// Mitsubishi GX Works2 project: Project   PLC: Q03UDV

PROGRAM MAIN
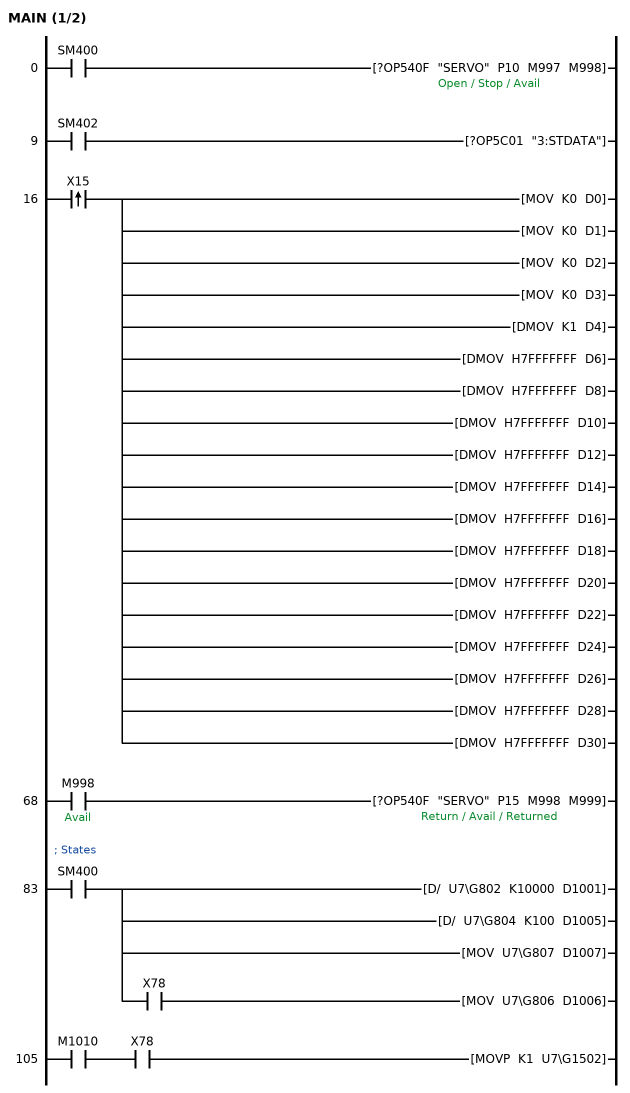
0     LD      SM400
      ?OP540F "SERVO" P10 M997 M998  ; Open / Stop / Avail
9     LD      SM402
      ?OP5C01 "3:STDATA"
16    LDP     X15
      MOV     K0 D0
      MOV     K0 D1
      MOV     K0 D2
      MOV     K0 D3
      DMOV    K1 D4
      DMOV    H7FFFFFFF D6
      DMOV    H7FFFFFFF D8
      DMOV    H7FFFFFFF D10
      DMOV    H7FFFFFFF D12
      DMOV    H7FFFFFFF D14
      DMOV    H7FFFFFFF D16
      DMOV    H7FFFFFFF D18
      DMOV    H7FFFFFFF D20
      DMOV    H7FFFFFFF D22
      DMOV    H7FFFFFFF D24
      DMOV    H7FFFFFFF D26
      DMOV    H7FFFFFFF D28
      DMOV    H7FFFFFFF D30
68    LD      M998  ; Avail
      ?OP540F "SERVO" P15 M998 M999  ; Return / Returned
; States
83    LD      SM400
      D/      U7\G802 K10000 D1001
      D/      U7\G804 K100 D1005
      MOV     U7\G807 D1007
      AND     X78
      MOV     U7\G806 D1006
105   LD      M1010
      AND     X78
      MOVP    K1 U7\G1502
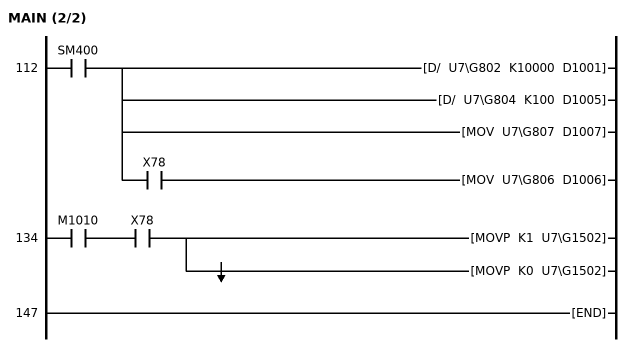
112   LD      SM400
      D/      U7\G802 K10000 D1001
      D/      U7\G804 K100 D1005
      MOV     U7\G807 D1007
      AND     X78
      MOV     U7\G806 D1006
134   LD      M1010
      AND     X78
      MOVP    K1 U7\G1502
      MEF
      MOVP    K0 U7\G1502
147   END
END_PROGRAM

PROGRAM SERVO
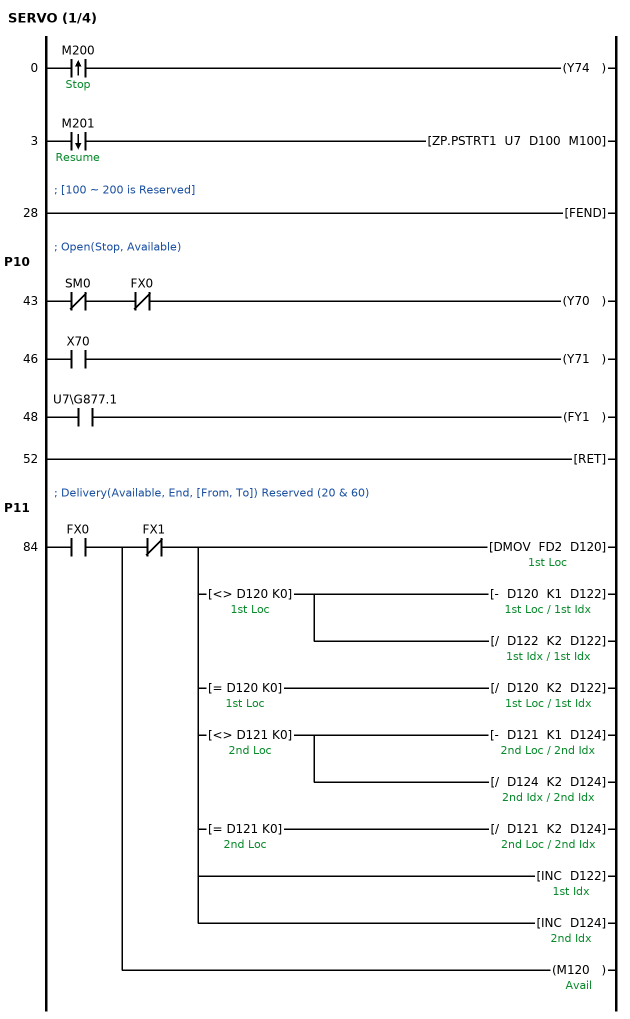
0     LDP     M200  ; Stop
      OUT     Y74
3     LDF     M201  ; Resume
      ZP.PSTRT1 U7 D100 M100
; [100 ~ 200 is Reserved]
28    FEND
      P10
; Open(Stop, Available)
43    LDI     SM0
      ANI     FX0
      OUT     Y70
46    LD      X70
      OUT     Y71
48    LD      U7\G877.1
      OUT     FY1
52    RET
      P11
; Delivery(Available, End, [From, To]) Reserved (20 & 60)
84    LD      FX0
      MPS
      ANI     FX1
      DMOV    FD2 D120  ; 1st Loc
      MPS
      AND<>   D120 K0  ; 1st Loc
      -       D120 K1 D122  ; 1st Idx
      /       D122 K2 D122
      MRD
      AND=    D120 K0  ; 1st Loc
      /       D120 K2 D122
      MRD
      AND<>   D121 K0  ; 2nd Loc
      -       D121 K1 D124  ; 2nd Idx
      /       D124 K2 D124
      MRD
      AND=    D121 K0  ; 2nd Loc
      /       D121 K2 D124
      MPP
      INC     D122
      INC     D124
      MPP
      OUT     M120  ; Avail
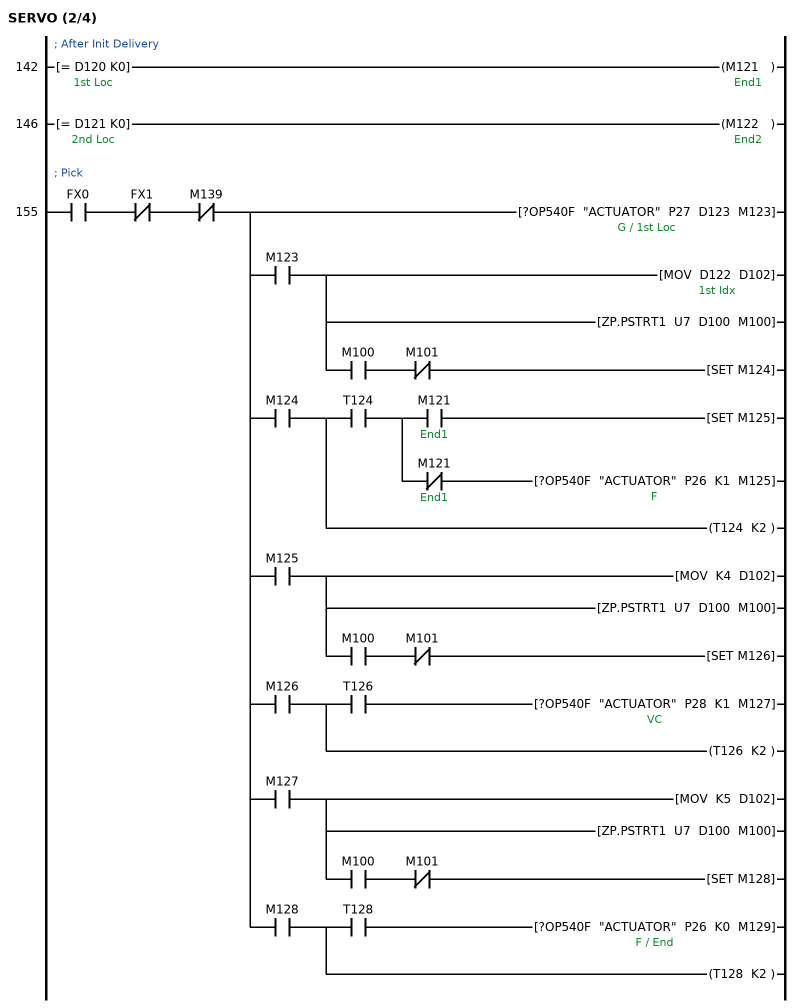
; After Init Delivery
142   LD=     D120 K0  ; 1st Loc
      OUT     M121  ; End1
146   LD=     D121 K0  ; 2nd Loc
      OUT     M122  ; End2
; Pick
155   LD      FX0
      ANI     FX1
      ANI     M139
      ?OP540F "ACTUATOR" P27 D123 M123  ; G / 1st Loc
      MPS
      AND     M123
      MOV     D122 D102
      ZP.PSTRT1 U7 D100 M100
      AND     M100
      ANI     M101
      SET     M124
      MRD
      AND     M124
      MPS
      AND     T124
      MPS
      AND     M121  ; End1
      SET     M125
      MPP
      ANI     M121  ; End1
      ?OP540F "ACTUATOR" P26 K1 M125  ; F
      MPP
      OUT     T124 K2
      MRD
      AND     M125
      MOV     K4 D102
      ZP.PSTRT1 U7 D100 M100
      AND     M100
      ANI     M101
      SET     M126
      MRD
      AND     M126
      MPS
      AND     T126
      ?OP540F "ACTUATOR" P28 K1 M127  ; VC
      MPP
      OUT     T126 K2
      MRD
      AND     M127
      MOV     K5 D102
      ZP.PSTRT1 U7 D100 M100
      AND     M100
      ANI     M101
      SET     M128
      MPP
      AND     M128
      MPS
      AND     T128
      ?OP540F "ACTUATOR" P26 K0 M129  ; End
      MPP
      OUT     T128 K2
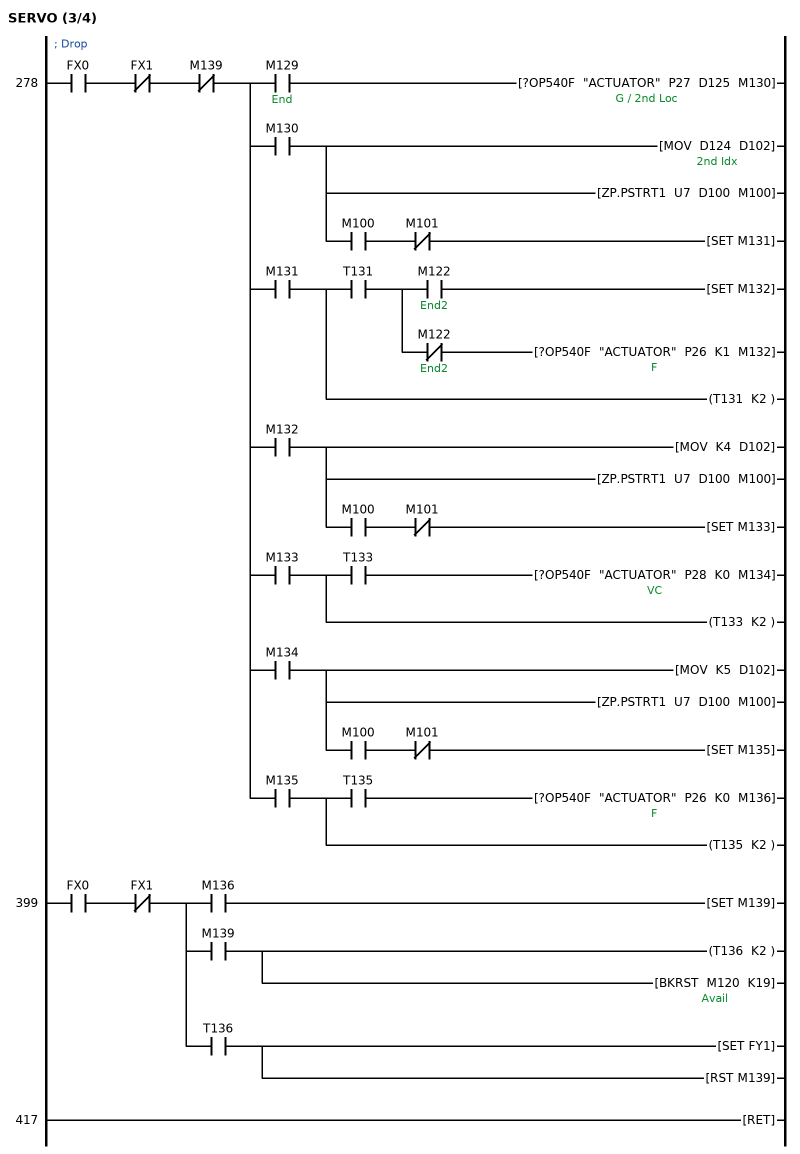
; Drop
278   LD      FX0
      ANI     FX1
      ANI     M139
      MPS
      AND     M129  ; End
      ?OP540F "ACTUATOR" P27 D125 M130  ; 2nd Loc
      MRD
      AND     M130
      MOV     D124 D102
      ZP.PSTRT1 U7 D100 M100
      AND     M100
      ANI     M101
      SET     M131
      MRD
      AND     M131
      MPS
      AND     T131
      MPS
      AND     M122  ; End2
      SET     M132
      MPP
      ANI     M122  ; End2
      ?OP540F "ACTUATOR" P26 K1 M132
      MPP
      OUT     T131 K2
      MRD
      AND     M132
      MOV     K4 D102
      ZP.PSTRT1 U7 D100 M100
      AND     M100
      ANI     M101
      SET     M133
      MRD
      AND     M133
      MPS
      AND     T133
      ?OP540F "ACTUATOR" P28 K0 M134
      MPP
      OUT     T133 K2
      MRD
      AND     M134
      MOV     K5 D102
      ZP.PSTRT1 U7 D100 M100
      AND     M100
      ANI     M101
      SET     M135
      MPP
      AND     M135
      MPS
      AND     T135
      ?OP540F "ACTUATOR" P26 K0 M136
      MPP
      OUT     T135 K2
399   LD      FX0
      ANI     FX1
      MPS
      AND     M136
      SET     M139
      MRD
      AND     M139
      OUT     T136 K2
      BKRST   M120 K19
      MPP
      AND     T136
      SET     FY1
      RST     M139
417   RET
      P15
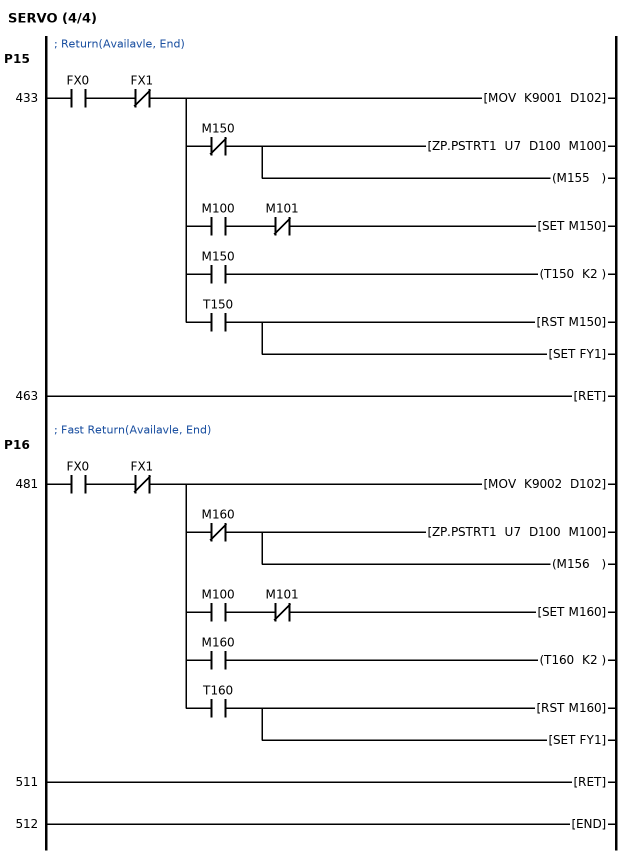
; Return(Availavle, End)
433   LD      FX0
      ANI     FX1
      MOV     K9001 D102
      MPS
      ANI     M150
      ZP.PSTRT1 U7 D100 M100
      OUT     M155
      MRD
      AND     M100
      ANI     M101
      SET     M150
      MRD
      AND     M150
      OUT     T150 K2
      MPP
      AND     T150
      RST     M150
      SET     FY1
463   RET
      P16
; Fast Return(Availavle, End)
481   LD      FX0
      ANI     FX1
      MOV     K9002 D102
      MPS
      ANI     M160
      ZP.PSTRT1 U7 D100 M100
      OUT     M156
      MRD
      AND     M100
      ANI     M101
      SET     M160
      MRD
      AND     M160
      OUT     T160 K2
      MPP
      AND     T160
      RST     M160
      SET     FY1
511   RET
512   END
END_PROGRAM

PROGRAM ACTUATOR
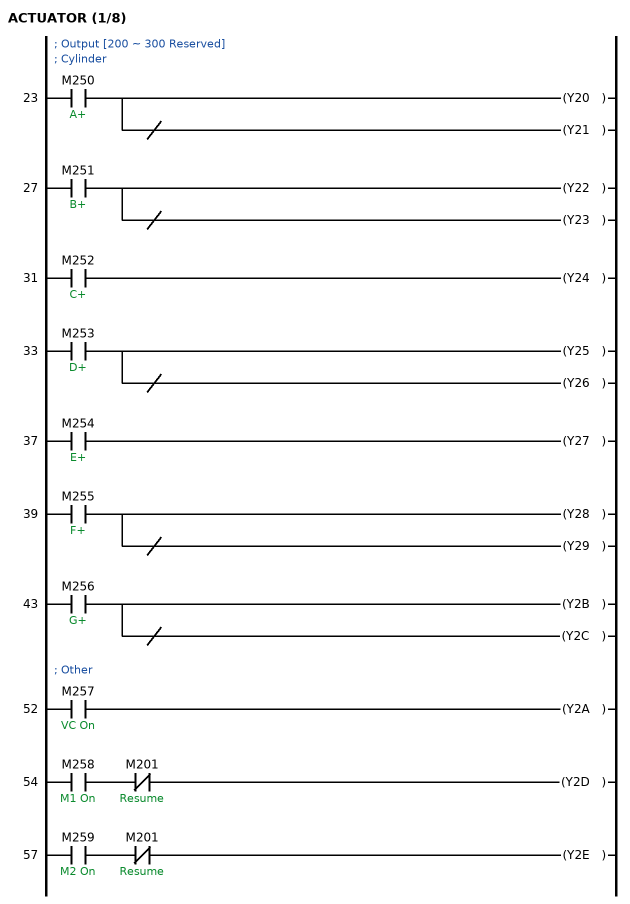
; Output [200 ~ 300 Reserved]
; Cylinder
23    LD      M250  ; A+
      OUT     Y20
      INV
      OUT     Y21
27    LD      M251  ; B+
      OUT     Y22
      INV
      OUT     Y23
31    LD      M252  ; C+
      OUT     Y24
33    LD      M253  ; D+
      OUT     Y25
      INV
      OUT     Y26
37    LD      M254  ; E+
      OUT     Y27
39    LD      M255  ; F+
      OUT     Y28
      INV
      OUT     Y29
43    LD      M256  ; G+
      OUT     Y2B
      INV
      OUT     Y2C
; Other
52    LD      M257  ; VC On
      OUT     Y2A
54    LD      M258  ; M1 On
      ANI     M201  ; Resume
      OUT     Y2D
57    LD      M259  ; M2 On
      ANI     M201  ; Resume
      OUT     Y2E
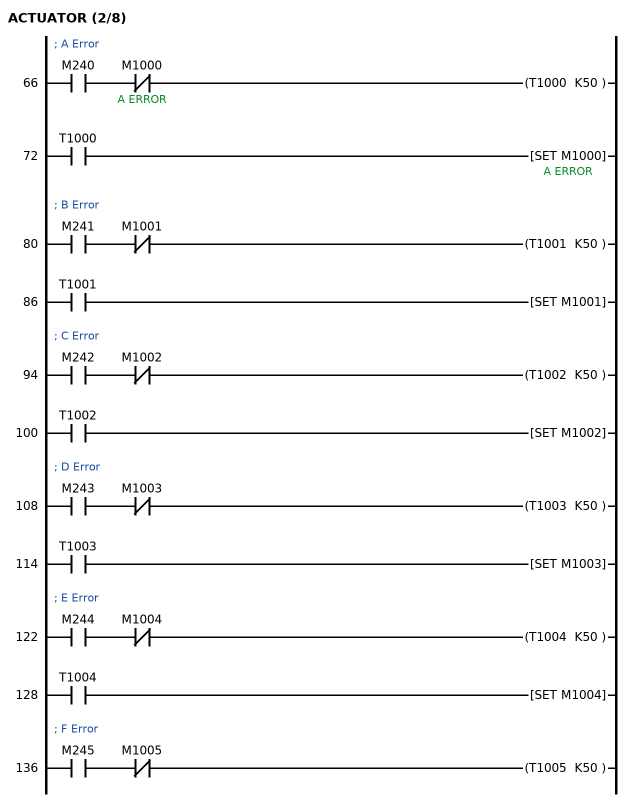
; A Error
66    LD      M240
      ANI     M1000  ; A ERROR
      OUT     T1000 K50
72    LD      T1000
      SET     M1000  ; A ERROR
; B Error
80    LD      M241
      ANI     M1001
      OUT     T1001 K50
86    LD      T1001
      SET     M1001
; C Error
94    LD      M242
      ANI     M1002
      OUT     T1002 K50
100   LD      T1002
      SET     M1002
; D Error
108   LD      M243
      ANI     M1003
      OUT     T1003 K50
114   LD      T1003
      SET     M1003
; E Error
122   LD      M244
      ANI     M1004
      OUT     T1004 K50
128   LD      T1004
      SET     M1004
; F Error
136   LD      M245
      ANI     M1005
      OUT     T1005 K50
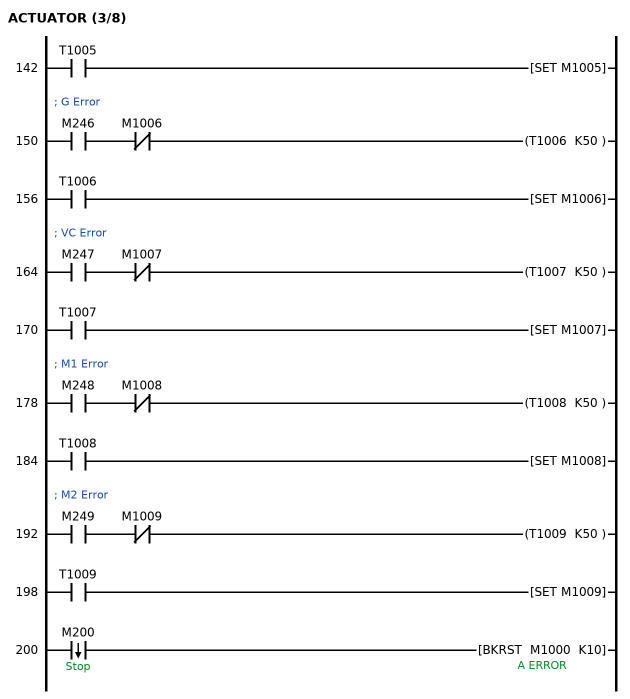
142   LD      T1005
      SET     M1005
; G Error
150   LD      M246
      ANI     M1006
      OUT     T1006 K50
156   LD      T1006
      SET     M1006
; VC Error
164   LD      M247
      ANI     M1007
      OUT     T1007 K50
170   LD      T1007
      SET     M1007
; M1 Error
178   LD      M248
      ANI     M1008
      OUT     T1008 K50
184   LD      T1008
      SET     M1008
; M2 Error
192   LD      M249
      ANI     M1009
      OUT     T1009 K50
198   LD      T1009
      SET     M1009
200   LDF     M200  ; Stop
      BKRST   M1000 K10
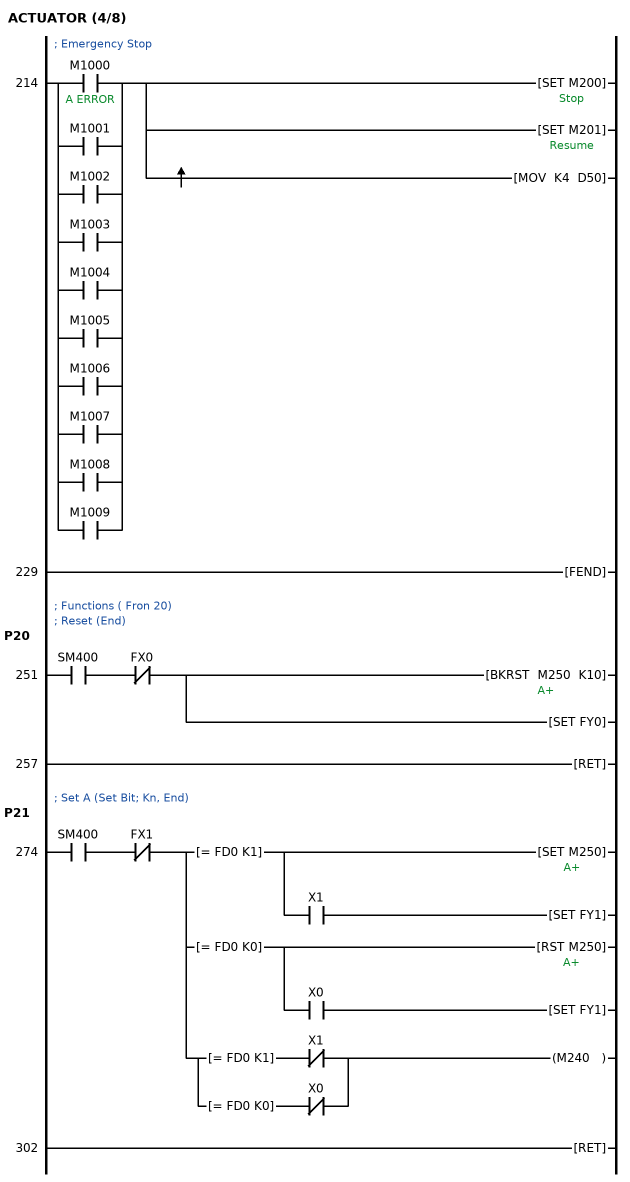
; Emergency Stop
214   LD      M1000  ; A ERROR
      OR      M1001
      OR      M1002
      OR      M1003
      OR      M1004
      OR      M1005
      OR      M1006
      OR      M1007
      OR      M1008
      OR      M1009
      SET     M200  ; Stop
      SET     M201  ; Resume
      MEP
      MOV     K4 D50
229   FEND
; Functions ( Fron 20)
      P20
; Reset (End)
251   LD      SM400
      ANI     FX0
      BKRST   M250 K10
      SET     FY0
257   RET
      P21
; Set A (Set Bit; Kn, End)
274   LD      SM400
      ANI     FX1
      MPS
      AND=    FD0 K1
      SET     M250  ; A+
      AND     X1
      SET     FY1
      MRD
      AND=    FD0 K0
      RST     M250  ; A+
      AND     X0
      SET     FY1
      MPP
      LD=     FD0 K1
      ANI     X1
      LD=     FD0 K0
      ANI     X0
      ORB
      ANB
      OUT     M240
302   RET
      P22
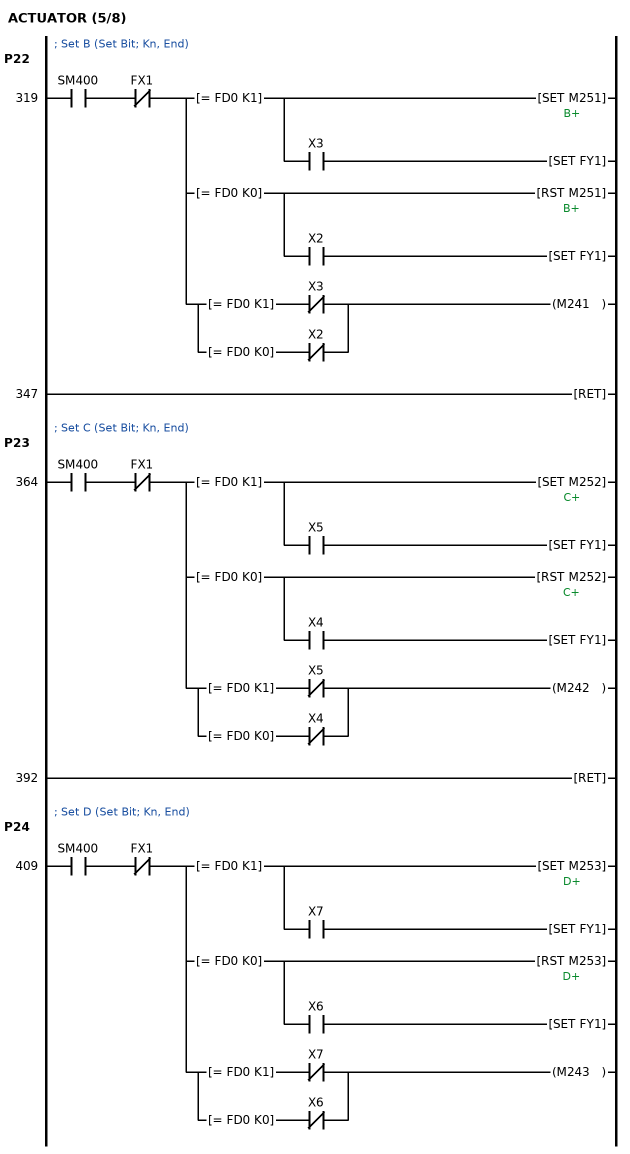
; Set B (Set Bit; Kn, End)
319   LD      SM400
      ANI     FX1
      MPS
      AND=    FD0 K1
      SET     M251  ; B+
      AND     X3
      SET     FY1
      MRD
      AND=    FD0 K0
      RST     M251  ; B+
      AND     X2
      SET     FY1
      MPP
      LD=     FD0 K1
      ANI     X3
      LD=     FD0 K0
      ANI     X2
      ORB
      ANB
      OUT     M241
347   RET
      P23
; Set C (Set Bit; Kn, End)
364   LD      SM400
      ANI     FX1
      MPS
      AND=    FD0 K1
      SET     M252  ; C+
      AND     X5
      SET     FY1
      MRD
      AND=    FD0 K0
      RST     M252  ; C+
      AND     X4
      SET     FY1
      MPP
      LD=     FD0 K1
      ANI     X5
      LD=     FD0 K0
      ANI     X4
      ORB
      ANB
      OUT     M242
392   RET
      P24
; Set D (Set Bit; Kn, End)
409   LD      SM400
      ANI     FX1
      MPS
      AND=    FD0 K1
      SET     M253  ; D+
      AND     X7
      SET     FY1
      MRD
      AND=    FD0 K0
      RST     M253  ; D+
      AND     X6
      SET     FY1
      MPP
      LD=     FD0 K1
      ANI     X7
      LD=     FD0 K0
      ANI     X6
      ORB
      ANB
      OUT     M243
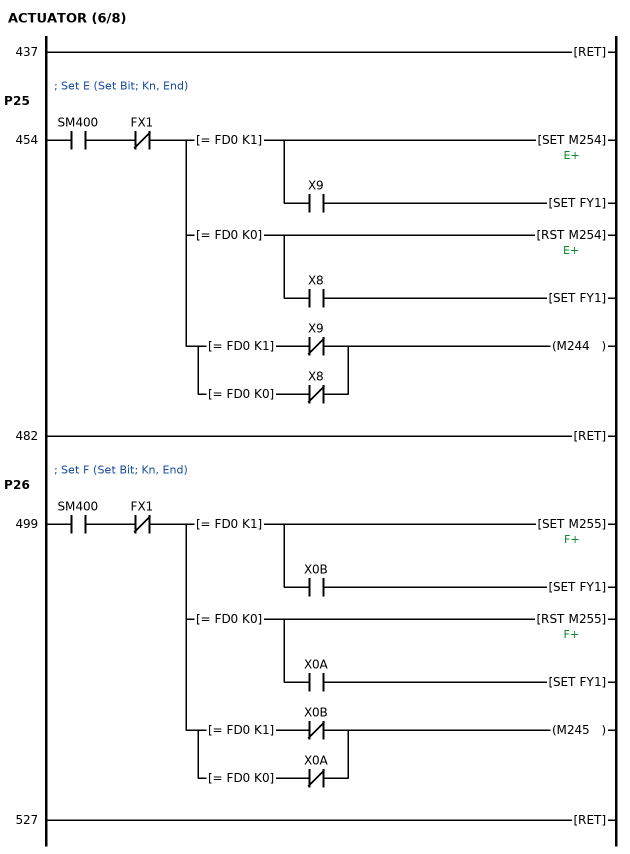
437   RET
      P25
; Set E (Set Bit; Kn, End)
454   LD      SM400
      ANI     FX1
      MPS
      AND=    FD0 K1
      SET     M254  ; E+
      AND     X9
      SET     FY1
      MRD
      AND=    FD0 K0
      RST     M254  ; E+
      AND     X8
      SET     FY1
      MPP
      LD=     FD0 K1
      ANI     X9
      LD=     FD0 K0
      ANI     X8
      ORB
      ANB
      OUT     M244
482   RET
      P26
; Set F (Set Bit; Kn, End)
499   LD      SM400
      ANI     FX1
      MPS
      AND=    FD0 K1
      SET     M255  ; F+
      AND     X0B
      SET     FY1
      MRD
      AND=    FD0 K0
      RST     M255  ; F+
      AND     X0A
      SET     FY1
      MPP
      LD=     FD0 K1
      ANI     X0B
      LD=     FD0 K0
      ANI     X0A
      ORB
      ANB
      OUT     M245
527   RET
      P27
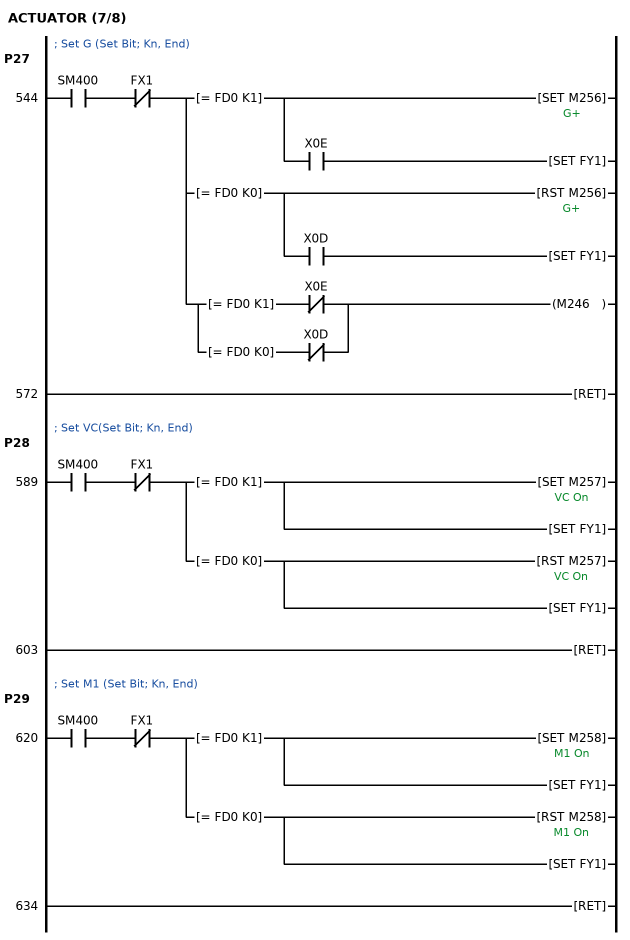
; Set G (Set Bit; Kn, End)
544   LD      SM400
      ANI     FX1
      MPS
      AND=    FD0 K1
      SET     M256  ; G+
      AND     X0E
      SET     FY1
      MRD
      AND=    FD0 K0
      RST     M256  ; G+
      AND     X0D
      SET     FY1
      MPP
      LD=     FD0 K1
      ANI     X0E
      LD=     FD0 K0
      ANI     X0D
      ORB
      ANB
      OUT     M246
572   RET
      P28
; Set VC(Set Bit; Kn, End)
589   LD      SM400
      ANI     FX1
      MPS
      AND=    FD0 K1
      SET     M257  ; VC On
      SET     FY1
      MPP
      AND=    FD0 K0
      RST     M257  ; VC On
      SET     FY1
603   RET
      P29
; Set M1 (Set Bit; Kn, End)
620   LD      SM400
      ANI     FX1
      MPS
      AND=    FD0 K1
      SET     M258  ; M1 On
      SET     FY1
      MPP
      AND=    FD0 K0
      RST     M258  ; M1 On
      SET     FY1
634   RET
      P30
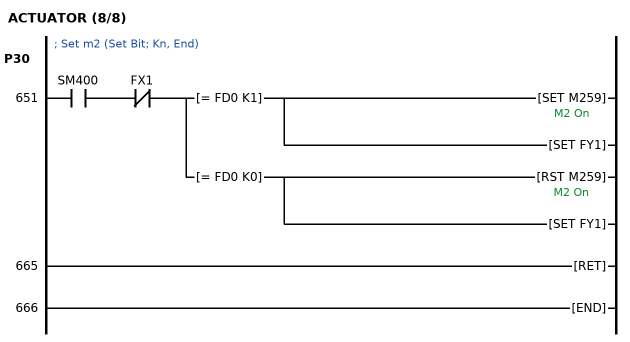
; Set m2 (Set Bit; Kn, End)
651   LD      SM400
      ANI     FX1
      MPS
      AND=    FD0 K1
      SET     M259  ; M2 On
      SET     FY1
      MPP
      AND=    FD0 K0
      RST     M259  ; M2 On
      SET     FY1
665   RET
666   END
END_PROGRAM

PROGRAM PART3
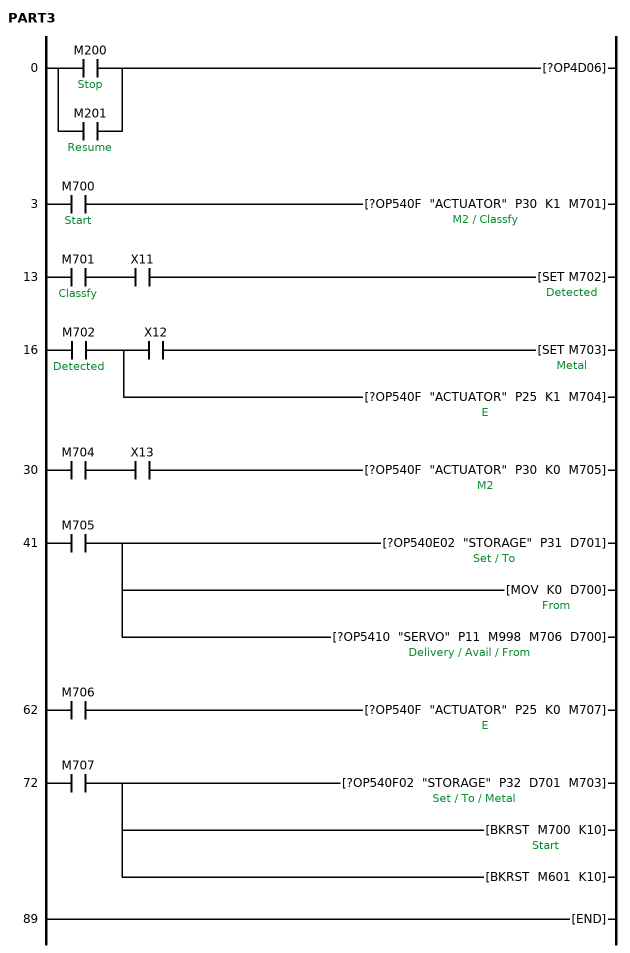
0     LD      M200  ; Stop
      OR      M201  ; Resume
      ?OP4D06
3     LD      M700  ; Start
      ?OP540F "ACTUATOR" P30 K1 M701  ; M2 / Classfy
13    LD      M701  ; Classfy
      AND     X11
      SET     M702  ; Detected
16    LD      M702  ; Detected
      MPS
      AND     X12
      SET     M703  ; Metal
      MPP
      ?OP540F "ACTUATOR" P25 K1 M704  ; E
30    LD      M704
      AND     X13
      ?OP540F "ACTUATOR" P30 K0 M705
41    LD      M705
      ?OP540E02 "STORAGE" P31 D701  ; Set / To
      MOV     K0 D700  ; From
      ?OP5410 "SERVO" P11 M998 M706 D700  ; Delivery / Avail
62    LD      M706
      ?OP540F "ACTUATOR" P25 K0 M707
72    LD      M707
      ?OP540F02 "STORAGE" P32 D701 M703  ; Set
      BKRST   M700 K10
      BKRST   M601 K10
89    END
END_PROGRAM

PROGRAM STORAGE
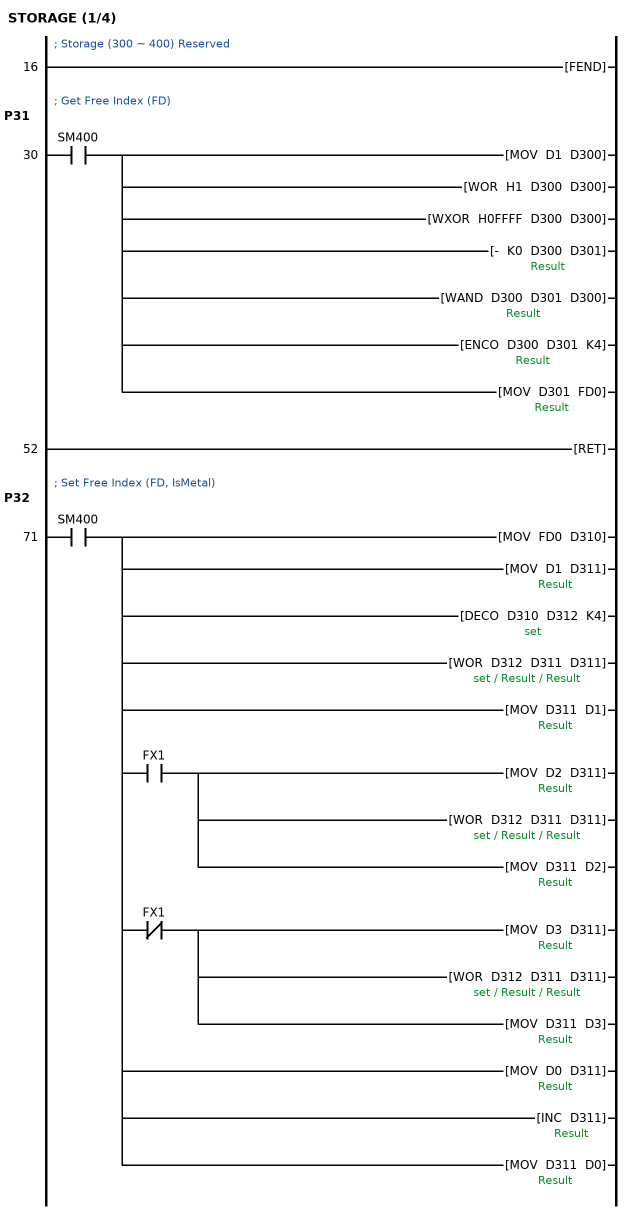
; Storage (300 ~ 400) Reserved
16    FEND
      P31
; Get Free Index (FD)
30    LD      SM400
      MOV     D1 D300
      WOR     H1 D300 D300
      WXOR    H0FFFF D300 D300
      -       K0 D300 D301  ; Result
      WAND    D300 D301 D300
      ENCO    D300 D301 K4
      MOV     D301 FD0
52    RET
      P32
; Set Free Index (FD, IsMetal)
71    LD      SM400
      MOV     FD0 D310
      MOV     D1 D311  ; Result
      DECO    D310 D312 K4  ; set
      WOR     D312 D311 D311
      MOV     D311 D1
      MPS
      AND     FX1
      MOV     D2 D311
      WOR     D312 D311 D311
      MOV     D311 D2
      MRD
      ANI     FX1
      MOV     D3 D311
      WOR     D312 D311 D311
      MOV     D311 D3
      MPP
      MOV     D0 D311
      INC     D311
      MOV     D311 D0
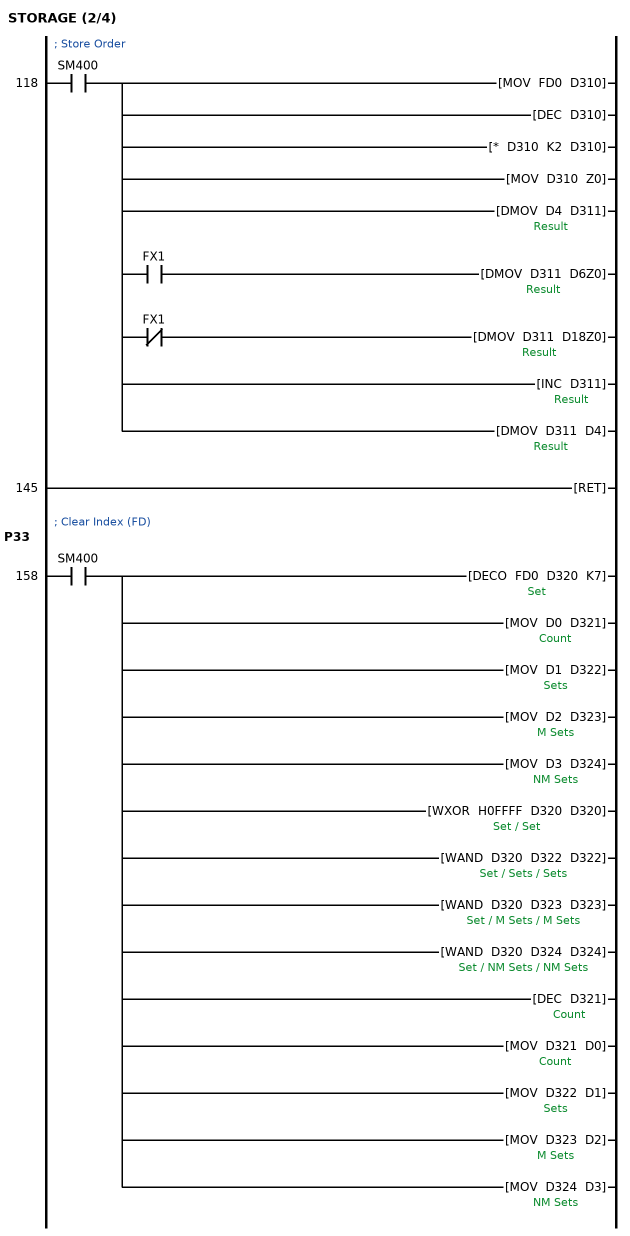
; Store Order
118   LD      SM400
      MOV     FD0 D310
      DEC     D310
      *       D310 K2 D310
      MOV     D310 Z0
      DMOV    D4 D311
      MPS
      AND     FX1
      DMOV    D311 D6Z0
      MRD
      ANI     FX1
      DMOV    D311 D18Z0
      MPP
      INC     D311
      DMOV    D311 D4
145   RET
      P33
; Clear Index (FD)
158   LD      SM400
      DECO    FD0 D320 K7  ; Set
      MOV     D0 D321  ; Count
      MOV     D1 D322  ; Sets
      MOV     D2 D323  ; M Sets
      MOV     D3 D324  ; NM Sets
      WXOR    H0FFFF D320 D320
      WAND    D320 D322 D322
      WAND    D320 D323 D323
      WAND    D320 D324 D324
      DEC     D321
      MOV     D321 D0
      MOV     D322 D1
      MOV     D323 D2
      MOV     D324 D3
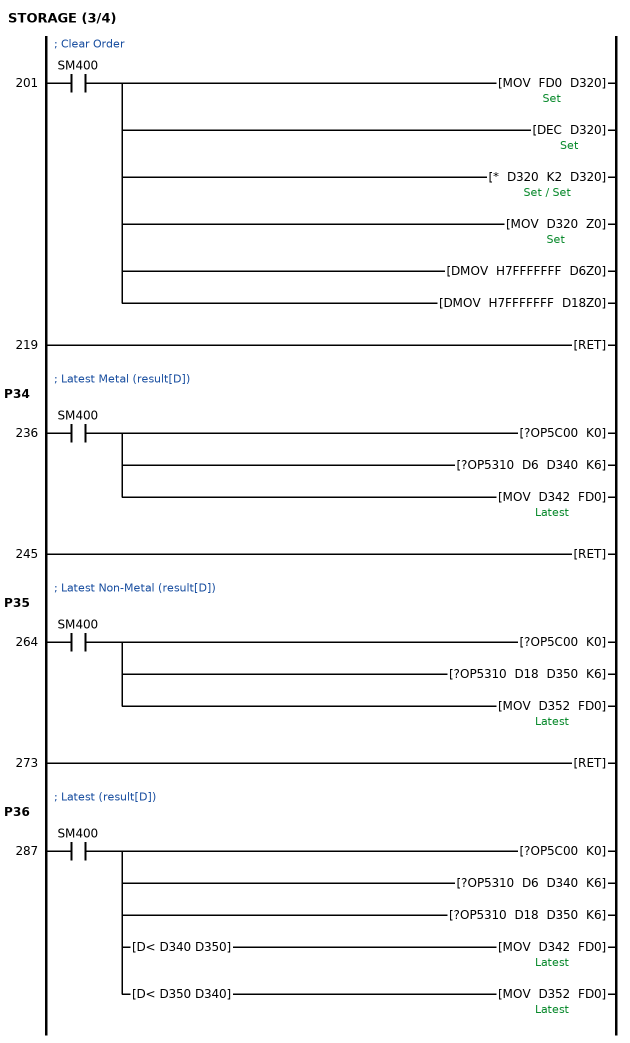
; Clear Order
201   LD      SM400
      MOV     FD0 D320
      DEC     D320
      *       D320 K2 D320
      MOV     D320 Z0
      DMOV    H7FFFFFFF D6Z0
      DMOV    H7FFFFFFF D18Z0
219   RET
      P34
; Latest Metal (result[D])
236   LD      SM400
      ?OP5C00 K0
      ?OP5310 D6 D340 K6
      MOV     D342 FD0  ; Latest
245   RET
      P35
; Latest Non-Metal (result[D])
264   LD      SM400
      ?OP5C00 K0
      ?OP5310 D18 D350 K6
      MOV     D352 FD0  ; Latest
273   RET
      P36
; Latest (result[D])
287   LD      SM400
      ?OP5C00 K0
      ?OP5310 D6 D340 K6
      ?OP5310 D18 D350 K6
      MPS
      ANDD<   D340 D350
      MOV     D342 FD0
      MPP
      ANDD<   D350 D340
      MOV     D352 FD0
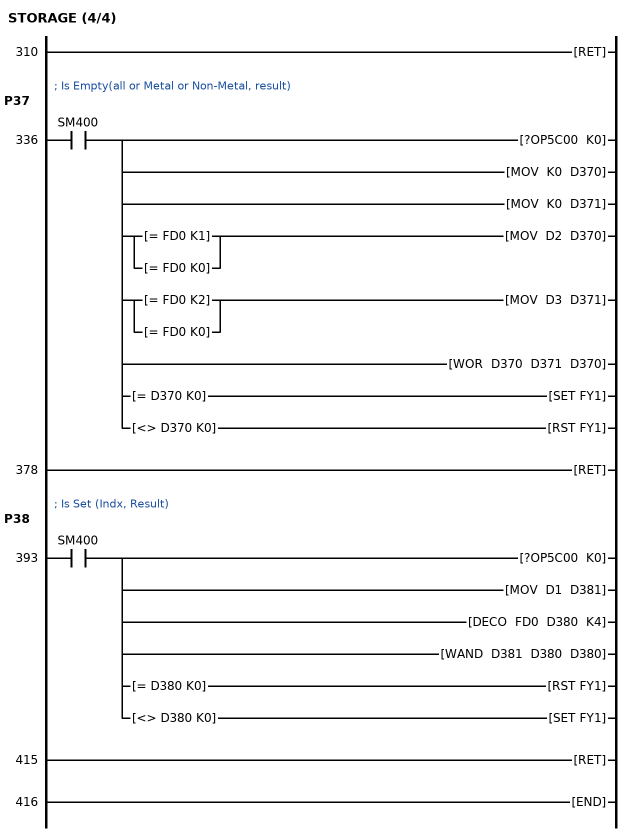
310   RET
      P37
; Is Empty(all or Metal or Non-Metal, result)
336   LD      SM400
      ?OP5C00 K0
      MOV     K0 D370
      MOV     K0 D371
      MPS
      LD=     FD0 K1
      OR=     FD0 K0
      ANB
      MOV     D2 D370
      MRD
      LD=     FD0 K2
      OR=     FD0 K0
      ANB
      MOV     D3 D371
      MPP
      WOR     D370 D371 D370
      MPS
      AND=    D370 K0
      SET     FY1
      MPP
      AND<>   D370 K0
      RST     FY1
378   RET
      P38
; Is Set (Indx, Result)
393   LD      SM400
      ?OP5C00 K0
      MOV     D1 D381
      DECO    FD0 D380 K4
      WAND    D381 D380 D380
      MPS
      AND=    D380 K0
      RST     FY1
      MPP
      AND<>   D380 K0
      SET     FY1
415   RET
416   END
END_PROGRAM

PROGRAM PART1
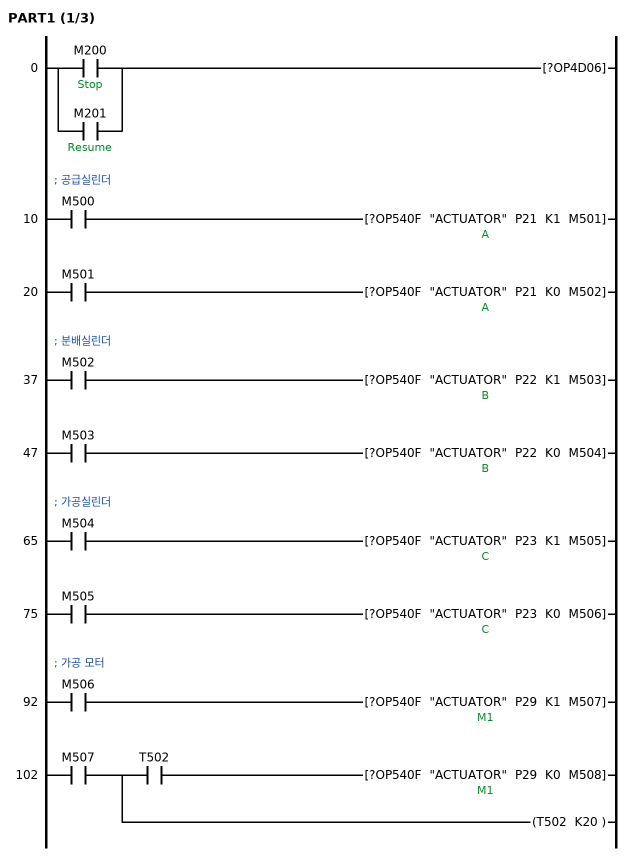
0     LD      M200  ; Stop
      OR      M201  ; Resume
      ?OP4D06
; 공급실린더
10    LD      M500
      ?OP540F "ACTUATOR" P21 K1 M501  ; A
20    LD      M501
      ?OP540F "ACTUATOR" P21 K0 M502
; 분배실린더
37    LD      M502
      ?OP540F "ACTUATOR" P22 K1 M503  ; B
47    LD      M503
      ?OP540F "ACTUATOR" P22 K0 M504
; 가공실린더
65    LD      M504
      ?OP540F "ACTUATOR" P23 K1 M505  ; C
75    LD      M505
      ?OP540F "ACTUATOR" P23 K0 M506
; 가공 모터
92    LD      M506
      ?OP540F "ACTUATOR" P29 K1 M507  ; M1
102   LD      M507
      MPS
      AND     T502
      ?OP540F "ACTUATOR" P29 K0 M508
      MPP
      OUT     T502 K20
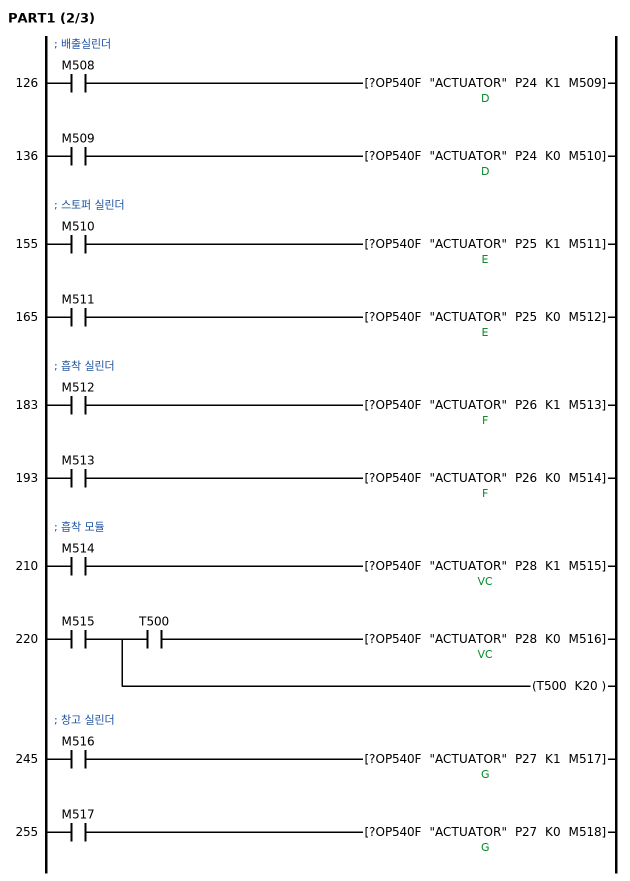
; 배출실린더
126   LD      M508
      ?OP540F "ACTUATOR" P24 K1 M509  ; D
136   LD      M509
      ?OP540F "ACTUATOR" P24 K0 M510
; 스토퍼 실린더
155   LD      M510
      ?OP540F "ACTUATOR" P25 K1 M511  ; E
165   LD      M511
      ?OP540F "ACTUATOR" P25 K0 M512
; 흡착 실린더
183   LD      M512
      ?OP540F "ACTUATOR" P26 K1 M513  ; F
193   LD      M513
      ?OP540F "ACTUATOR" P26 K0 M514
; 흡착 모듈
210   LD      M514
      ?OP540F "ACTUATOR" P28 K1 M515  ; VC
220   LD      M515
      MPS
      AND     T500
      ?OP540F "ACTUATOR" P28 K0 M516
      MPP
      OUT     T500 K20
; 창고 실린더
245   LD      M516
      ?OP540F "ACTUATOR" P27 K1 M517  ; G
255   LD      M517
      ?OP540F "ACTUATOR" P27 K0 M518
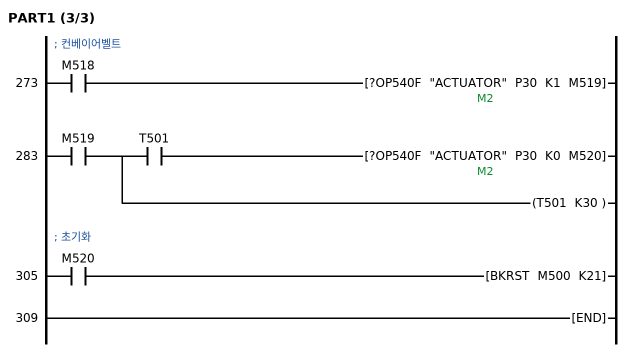
; 컨베이어벨트
273   LD      M518
      ?OP540F "ACTUATOR" P30 K1 M519  ; M2
283   LD      M519
      MPS
      AND     T501
      ?OP540F "ACTUATOR" P30 K0 M520
      MPP
      OUT     T501 K30
; 초기화
305   LD      M520
      BKRST   M500 K21
309   END
END_PROGRAM

PROGRAM PART2
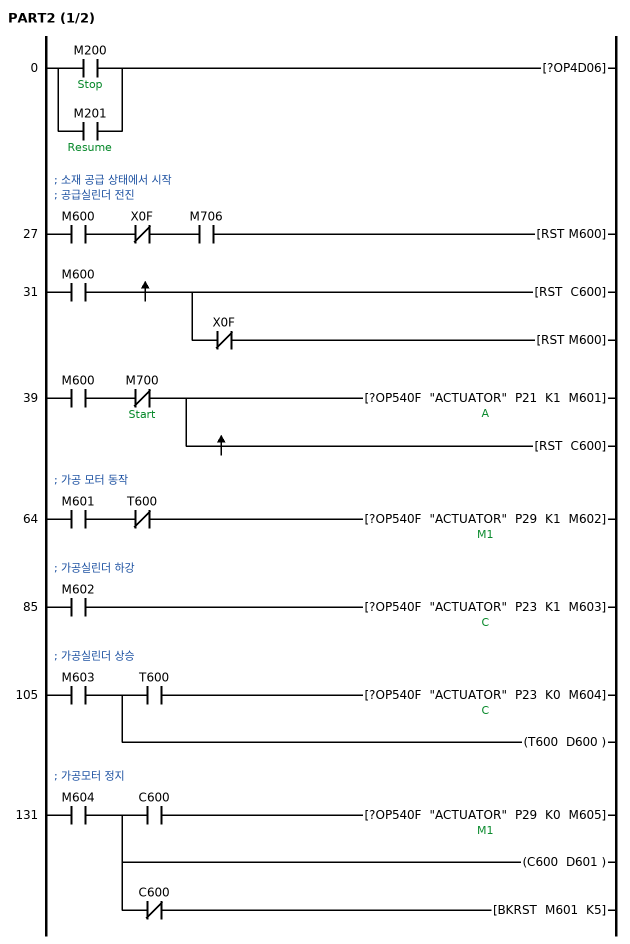
0     LD      M200  ; Stop
      OR      M201  ; Resume
      ?OP4D06
; 소재 공급 상태에서 시작
; 공급실린더 전진
27    LD      M600
      ANI     X0F
      AND     M706
      RST     M600
31    LD      M600
      MEP
      RST     C600
      ANI     X0F
      RST     M600
39    LD      M600
      ANI     M700  ; Start
      ?OP540F "ACTUATOR" P21 K1 M601  ; A
      MEP
      RST     C600
; 가공 모터 동작
64    LD      M601
      ANI     T600
      ?OP540F "ACTUATOR" P29 K1 M602  ; M1
; 가공실린더 하강
85    LD      M602
      ?OP540F "ACTUATOR" P23 K1 M603  ; C
; 가공실린더 상승
105   LD      M603
      MPS
      AND     T600
      ?OP540F "ACTUATOR" P23 K0 M604
      MPP
      OUT     T600 D600
; 가공모터 정지
131   LD      M604
      MPS
      AND     C600
      ?OP540F "ACTUATOR" P29 K0 M605
      MPP
      OUT     C600 D601
      ANI     C600
      BKRST   M601 K5
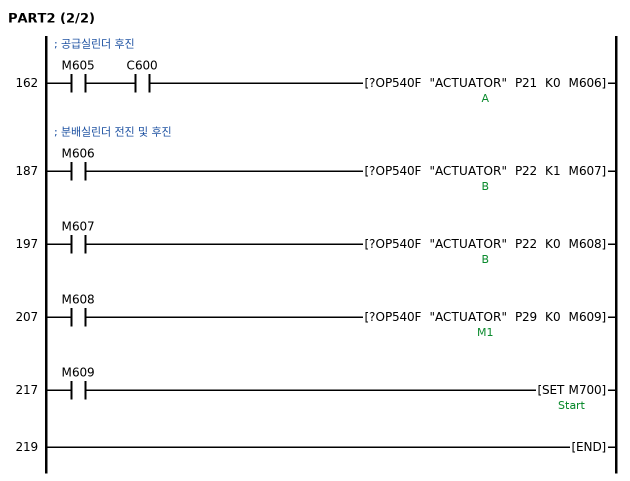
; 공급실린더 후진
162   LD      M605
      AND     C600
      ?OP540F "ACTUATOR" P21 K0 M606
; 분배실린더 전진 및 후진
187   LD      M606
      ?OP540F "ACTUATOR" P22 K1 M607  ; B
197   LD      M607
      ?OP540F "ACTUATOR" P22 K0 M608
207   LD      M608
      ?OP540F "ACTUATOR" P29 K0 M609
217   LD      M609
      SET     M700  ; Start
219   END
END_PROGRAM

PROGRAM PART4
